ABB RAPID module: Ecosystem_BASE.sysx

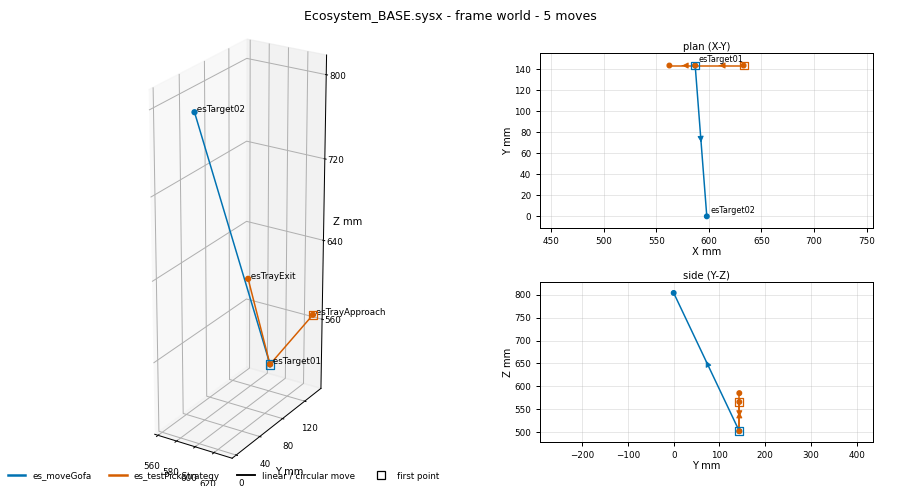
[picture p0: tool path of Ecosystem_BASE.sysx in frame world, 5 of 7 moves have a stored position in this frame; points joined in program order, loops and branches not executed]
MODULE Ecosystem_BASE(SYSMODULE)

    PERS num esNumber:=50;
    LOCAL PERS string esString:="I am a string";
    TASK PERS bool esBool:=FALSE;

    PERS tooldata esTool:=[TRUE,[[0,0,100],[1,0,0,0]],[0.1,[0,0,0.1],[1,0,0,0],0,0,0]];
    PERS wobjdata esWobj:=[FALSE,TRUE,"ROB_1",[[587.405,-129.894,406.227],[0.707718,-0.000019299,0.000021116,-0.706495]],[[0,0,0],[1,0,0,0]]];
    PERS wobjdata esWobjRotated:=[FALSE,TRUE,"ROB_1",[[587.405,-129.893,406.227],[0.694722446,0.135002675,-0.134767241,-0.693522019]],[[0,0,0],[1,0,0,0]]];

    PERS robtarget esTarget01:=[[586.9355,143.4633,501.8817],[0.06600141,-0.009778698,-0.9976442,-0.01594038],[0,0,0,0],[9E+09,9E+09,9E+09,9E+09,9E+09,9E+09]];
    PERS robtarget esTarget02:=[[597.986,0,804.151],[0.382683,0,0.92388,0],[0,0,0,0],[9E+9,9E+9,9E+9,9E+9,9E+9,9E+9]];

    PERS robtarget esTray01:=[[586.9355,143.4633,501.8817],[0.06600141,-0.009778698,-0.9976442,-0.01594038],[0,0,0,0],[9E+09,9E+09,9E+09,9E+09,9E+09,9E+09]];
    PERS robtarget esTray02:=[[586.9352,-173.2587,501.8815],[0.06600121,-0.009778861,-0.9976443,-0.01594038],[-1,-1,-1,0],[9E+09,9E+09,9E+09,9E+09,9E+09,9E+09]];
    PERS robtarget esTray03:=[[362.377,-173.258,501.881],[0.0660002,-0.0097793,-0.997644,-0.0159399],[-1,-1,-1,0],[9E+9,9E+9,9E+9,9E+9,9E+9,9E+9]];
    PERS robtarget esTray04:=[[742.687,-88.3141,577.45],[0.330698,0.0538063,0.942112,-0.0129992],[-1,0,-1,0],[9E+9,9E+9,9E+9,9E+9,9E+9,9E+9]];

    PERS robtarget esTrayGrip:=[[586.935,143.463,501.882],[0.0660014,-0.0097787,-0.997644,-0.0159404],[0,0,0,0],[9E+9,9E+9,9E+9,9E+9,9E+9,9E+9]];
    PERS robtarget esTrayApproach:=[[633.01,143.463,565.772],[0.0660018,-0.00977868,-0.997644,-0.0159404],[0,0,0,0],[9E+9,9E+9,9E+9,9E+9,9E+9,9E+9]];
    PERS robtarget esTrayExit:=[[562.396,143.463,585.147],[0.0660015,-0.00977873,-0.997644,-0.0159403],[0,0,0,0],[9E+9,9E+9,9E+9,9E+9,9E+9,9E+9]];

    PERS num esNumParts:=40;
    PERS num esNumRows:=11;
    PERS num esNumCols:=9;
    PERS num esCurrentPart:=3;
    PERS dnum esDNumValue:=4;
    PERS bool esSim:=TRUE;
    PERS num esArray{4}:=[1,2,3,4];
    PERS num esArray2D{4,2}:=[[1,2],[3,4],[5,8],[7,8]];

    CONST num pi:=3.1416;
    PERS pos esPose:=[100,200,300];
    PERS jointtarget esHome:=[[0,0,0,0,45,0],[9E+09,9E+09,9E+09,9E+09,9E+09,9E+09]];

    PROC es_Procedure_01()
        TPWrite "Ecosystem module procedure 1 called...";
    ENDPROC

    PROC es_Procedure_02()
        TPWrite "Ecosystem module procedure 2 called...";
    ENDPROC

    PROC es_moveGofa()
        MoveAbsJ esHome\NoEOffs,v100,z50,tool0\WObj:=wobj0;
        MoveL esTarget01,v100,z50,tool0\WObj:=wobj0;
        MoveL esTarget02,v100,z50,tool0\WObj:=wobj0;
        MoveAbsJ esHome\NoEOffs,v100,z50,tool0\WObj:=wobj0;
    ENDPROC

    PROC es_testPickStrategy()
        MoveL esTrayApproach,v100,z50,esTool\WObj:=wobj0;
        MoveL esTrayGrip,v50,fine,esTool\WObj:=wobj0;
        WaitTime 1;
        MoveL esTrayExit,v100,fine,esTool\WObj:=wobj0;
    ENDPROC
ENDMODULE
